PROGRAM Alias
VAR
END_VAR

//R1 & R2 : MCP**  
	//DI
	MCP_IO.MasterStopPB_Pressed					:= NOT Input.R1_01_00;  //NC - Master stop PB not pressed - black pb on mcp
	MCP_IO.CageEstopCircuitOK					:= Input.R1_01_01;  //case Estop circuit okay (Rly1 (120vac)
	MCP_IO.AutoModeSelected						:= Input.R1_01_02; // 0 = manual, 1=auto
	MCP_IO.PSU1_DCOK							:= Input.R1_01_03; //psu1 dc ok
	MCP_IO.MachineGNDrlyOpen					:= Input.R1_01_04; // machine ground lifted (opto board)	
	MCP_IO.CloseAllChargeRlyCommand				:= Input.R1_01_05; // command from screen room (opto)
	MCP_IO.OpenAllDumpRelayCommand				:= Input.R1_01_06; // command from screen room (opto)
	
	MCP_IO.Charger[1].inhibited					:= Input.R1_02_00; //TDK802 1
	MCP_IO.Charger[1].EndOfCharge				:= Input.R1_02_01; //TDK802 1
	MCP_IO.Charger[1].HV_isON					:= Input.R1_02_02; //TDK802 1
	MCP_IO.Charger[1].OverTemp					:= Input.R1_02_03; //TDK802 1
	MCP_IO.Charger[1].InterlockOpen				:= Input.R1_02_04; //TDK802 1
	MCP_IO.Charger[1].LoadFaulted				:= Input.R1_02_05; //TDK802 1
	MCP_IO.Charger[1].SummaryFaulted			:= Input.R1_02_06; //TDK802 1
	
	MCP_IO.Charger[2].inhibited					:= Input.R1_03_00; //TDK802 2
	MCP_IO.Charger[2].EndOfCharge				:= Input.R1_03_01; 
	MCP_IO.Charger[2].HV_isON					:= Input.R1_03_02; 
	MCP_IO.Charger[2].OverTemp					:= Input.R1_03_03; 
	MCP_IO.Charger[2].InterlockOpen				:= Input.R1_03_04; 
	MCP_IO.Charger[2].LoadFaulted				:= Input.R1_03_05; 
	MCP_IO.Charger[2].SummaryFaulted			:= Input.R1_03_06; 
	
	MCP_IO.Charger[3].inhibited					:= Input.R1_04_00; //TDK802 3
	MCP_IO.Charger[3].EndOfCharge				:= Input.R1_04_01; 
	MCP_IO.Charger[3].HV_isON					:= Input.R1_04_02; 
	MCP_IO.Charger[3].OverTemp					:= Input.R1_04_03; 
	MCP_IO.Charger[3].InterlockOpen				:= Input.R1_04_04; 
	MCP_IO.Charger[3].LoadFaulted				:= Input.R1_04_05; 
	MCP_IO.Charger[3].SummaryFaulted			:= Input.R1_04_06; 
	
	MCP_IO.Charger[4].inhibited					:= Input.R1_05_00; //TDK802 4
	MCP_IO.Charger[4].EndOfCharge				:= Input.R1_05_01; 
	MCP_IO.Charger[4].HV_isON					:= Input.R1_05_02; 
	MCP_IO.Charger[4].OverTemp					:= Input.R1_05_03; 
	MCP_IO.Charger[4].InterlockOpen				:= Input.R1_05_04; 
	MCP_IO.Charger[4].LoadFaulted				:= Input.R1_05_05; 
	MCP_IO.Charger[4].SummaryFaulted			:= Input.R1_05_06; 

	MCP_IO.Charger[5].inhibited					:= Input.R1_06_00; //TDK802 5
	MCP_IO.Charger[5].EndOfCharge				:= Input.R1_06_01; 
	MCP_IO.Charger[5].HV_isON					:= Input.R1_06_02; 
	MCP_IO.Charger[5].OverTemp					:= Input.R1_06_03; 
	MCP_IO.Charger[5].InterlockOpen				:= Input.R1_06_04; 
	MCP_IO.Charger[5].LoadFaulted				:= Input.R1_06_05; 
	MCP_IO.Charger[5].SummaryFaulted			:= Input.R1_06_06; 

	MCP_IO.Charger[6].inhibited					:= Input.R1_07_00; //TDK802 6
	MCP_IO.Charger[6].EndOfCharge				:= Input.R1_07_01; 
	MCP_IO.Charger[6].HV_isON					:= Input.R1_07_02; 
	MCP_IO.Charger[6].OverTemp					:= Input.R1_07_03; 
	MCP_IO.Charger[6].InterlockOpen				:= Input.R1_07_04; 
	MCP_IO.Charger[6].LoadFaulted				:= Input.R1_07_05; 
	MCP_IO.Charger[6].SummaryFaulted			:= Input.R1_07_06; 

	MCP_IO.Charger[7].inhibited					:= Input.R1_08_00; //TDK802 7
	MCP_IO.Charger[7].EndOfCharge				:= Input.R1_08_01; 
	MCP_IO.Charger[7].HV_isON					:= Input.R1_08_02; 
	MCP_IO.Charger[7].OverTemp					:= Input.R1_08_03; 
	MCP_IO.Charger[7].InterlockOpen				:= Input.R1_08_04; 
	MCP_IO.Charger[7].LoadFaulted				:= Input.R1_08_05; 
	MCP_IO.Charger[7].SummaryFaulted			:= Input.R1_08_06; 

	MCP_IO.Charger[8].inhibited					:= Input.R1_09_00; //TDK802 8
	MCP_IO.Charger[8].EndOfCharge				:= Input.R1_09_01; 
	MCP_IO.Charger[8].HV_isON					:= Input.R1_09_02; 
	MCP_IO.Charger[8].OverTemp					:= Input.R1_09_03; 
	MCP_IO.Charger[8].InterlockOpen				:= Input.R1_09_04; 
	MCP_IO.Charger[8].LoadFaulted				:= Input.R1_09_05; 
	MCP_IO.Charger[8].SummaryFaulted			:= Input.R1_09_06; 

	//AI
	MCP_IO.Charger[1].voltageFeedback_raw		:= Input.R2_03_00;
	MCP_IO.Charger[1].currentFeedback_raw		:= Input.R2_03_01;
	MCP_IO.Charger[2].voltageFeedback_raw		:= Input.R2_03_02;
	MCP_IO.Charger[2].currentFeedback_raw		:= Input.R2_03_03;
	MCP_IO.Charger[3].voltageFeedback_raw		:= Input.R2_03_04;
	MCP_IO.Charger[3].currentFeedback_raw		:= Input.R2_03_05;
	MCP_IO.Charger[4].voltageFeedback_raw		:= Input.R2_03_06;
	MCP_IO.Charger[4].currentFeedback_raw		:= Input.R2_03_07;
	MCP_IO.Charger[5].voltageFeedback_raw		:= Input.R2_04_00;
	MCP_IO.Charger[5].currentFeedback_raw		:= Input.R2_04_01;
	MCP_IO.Charger[6].voltageFeedback_raw		:= Input.R2_04_02;
	MCP_IO.Charger[6].currentFeedback_raw		:= Input.R2_04_03;
	MCP_IO.Charger[7].voltageFeedback_raw		:= Input.R2_04_04;
	MCP_IO.Charger[7].currentFeedback_raw		:= Input.R2_04_05;
	MCP_IO.Charger[8].voltageFeedback_raw		:= Input.R2_04_06;
	MCP_IO.Charger[8].currentFeedback_raw		:= Input.R2_04_07;
	
	//DQ
	Output.R2_01_00	:= MCP_IO.Charger[1].inhibit;
	Output.R2_01_01	:= MCP_IO.Charger[1].HV_ON;
	Output.R2_01_02	:= MCP_IO.Charger[2].inhibit;
	Output.R2_01_03	:= MCP_IO.Charger[2].HV_ON;
	Output.R2_01_04	:= MCP_IO.Charger[3].inhibit;
	Output.R2_01_05	:= MCP_IO.Charger[3].HV_ON;
	Output.R2_01_06	:= MCP_IO.Charger[4].inhibit;
	Output.R2_01_07	:= MCP_IO.Charger[4].HV_ON;
	
	Output.R2_02_00	:= MCP_IO.Charger[5].inhibit;
	Output.R2_02_01	:= MCP_IO.Charger[5].HV_ON;
	Output.R2_02_02	:= MCP_IO.Charger[6].inhibit;
	Output.R2_02_03	:= MCP_IO.Charger[6].HV_ON;
	Output.R2_02_04	:= MCP_IO.Charger[7].inhibit;
	Output.R2_02_05	:= MCP_IO.Charger[7].HV_ON;
	Output.R2_02_06	:= MCP_IO.Charger[8].inhibit;
	Output.R2_02_07	:= MCP_IO.Charger[8].HV_ON;
	
	Output.R2_06_00	:= MCP_IO.GLS1_hvON;
	Output.R2_06_01	:= MCP_IO.GLS2_hvON;
	Output.R2_06_02	:= MCP_IO.GLS3_hvON;
	Output.R2_06_03	:= MCP_IO.LiftMachineGND;
	Output.R2_06_04	:= MCP_IO.AllChargeRelaysClose; //only for slim
	Output.R2_06_05	:= MCP_IO.AllDumpRelaysOpen;  // only for slim
	
	//AQ
	Output.R2_05_00	:= MCP_IO.Charger[1].voltageSP;
	Output.R2_05_01	:= MCP_IO.Charger[2].voltageSP;
	Output.R2_05_02	:= MCP_IO.Charger[3].voltageSP;
	Output.R2_05_03	:= MCP_IO.Charger[4].voltageSP;	
	Output.R2_05_04	:= MCP_IO.Charger[5].voltageSP;
	Output.R2_05_05	:= MCP_IO.Charger[6].voltageSP;
	Output.R2_05_06	:= MCP_IO.Charger[7].voltageSP;
	Output.R2_05_07	:= MCP_IO.Charger[8].voltageSP;					
	
	Output.R2_07_00	:= MCP_IO.GLS1_voltageSP; //Form Trigger
	Output.R2_07_01	:= MCP_IO.GLS2_voltageSP;  //Preform trigger
	Output.R2_07_02	:= MCP_IO.GLS3_voltageSP; //preform cap charger

//R3 : Bank 1 (LCP1)***********************************************
	//EL3068 - AI
	LCP.Section[1].Peak.cap[1].voltageFeedback_raw := Input.R3_01_00;
	LCP.Section[1].Peak.cap[2].voltageFeedback_raw := Input.R3_01_01;
	LCP.Section[1].Peak.cap[3].voltageFeedback_raw := Input.R3_01_02;
	LCP.Section[1].Peak.cap[4].voltageFeedback_raw := Input.R3_01_03;
	LCP.Section[1].Peak.cap[5].voltageFeedback_raw := Input.R3_01_04;
	LCP.Section[1].Peak.cap[6].voltageFeedback_raw := Input.R3_01_05;
	LCP.Section[1].Peak.cap[7].voltageFeedback_raw := Input.R3_01_06;
	LCP.Section[1].Peak.cap[8].voltageFeedback_raw := Input.R3_01_07;
	LCP.Section[1].Peak.cap[9].voltageFeedback_raw := Input.R3_02_00;
	LCP.Section[1].Peak.cap[10].voltageFeedback_raw := Input.R3_02_01;
	
	LCP.Section[1].Sust.cap[1].voltageFeedback_raw := Input.R3_02_02;
	LCP.Section[1].Sust.cap[2].voltageFeedback_raw := Input.R3_02_03;
	
	//DI
	LCP.Section[1].Peak.ChargeRelay1_close 	:= Input.R3_03_00; //RLY 1A
	LCP.Section[1].Peak.ChargeRelay2_close 	:= Input.R3_03_01; //RLY 2A
	LCP.Section[1].Peak.DumpRelay1_close 	:= Input.R3_03_02; //RLY 3A
	LCP.Section[1].Peak.DumpRelay2_close	:= Input.R3_03_03; //RLY 4A
	LCP.Section[1].Sust.ChargeRelay1_close	:= Input.R3_03_04; //RLY 5A
	LCP.Section[1].Sust.ChargeRelay2_close	:= Input.R3_03_05; //RLY 6A
	LCP.Section[1].Sust.DumpRelay1_close	:= Input.R3_03_06; //RLY 7A
	LCP.Section[1].Sust.DumpRelay2_close	:= Input.R3_03_07; //RLY 8A
	
	LCP.Section[1].Peak.ShortContact1_close 	:= Input.R3_04_00; //psw1
	LCP.Section[1].Peak.UnshortContact1_close 	:= Input.R3_04_01; //psw2
	LCP.Section[1].Peak.ShortContact2_close 	:= Input.R3_04_02; //psw3
	LCP.Section[1].Peak.UnshortContact2_close 	:= Input.R3_04_03; //psw4
	LCP.Section[1].LossPneumaticPressure 		:= Input.R3_04_04; //psw5
	LCP.Section[1].PSU1_DCOK					:= Input.R3_04_05; //psu1 contact

	//DQ
	Output.R3_05_00 := LCP.Section[1].Peak.CloseChargeRelay1; //RLY1
	Output.R3_05_01 := LCP.Section[1].Peak.CloseChargeRelay2; //RLY2
	Output.R3_05_02 := LCP.Section[1].Peak.OpenDumpRelay1; //RLY3
	Output.R3_05_03 := LCP.Section[1].Peak.OpenDumpRelay2; //RLY4
	Output.R3_05_04 := LCP.Section[1].Sust.CloseChargeRelay1; //RLY5
	Output.R3_05_05 := LCP.Section[1].Sust.CloseChargeRelay2; //RLY6
	Output.R3_05_06 := LCP.Section[1].Sust.OpenDumpRelay1; //RLY7
	Output.R3_05_07 := LCP.Section[1].Sust.OpenDumpRelay2; //RLY8
	Output.R3_06_00 := LCP.Section[1].SystemReadyToCharge; //LED1

//R4 : Bank 2 (LCP2)***********************************************
	//EL3068 - AI
	LCP.Section[2].Peak.cap[1].voltageFeedback_raw := Input.R4_01_00;
	LCP.Section[2].Peak.cap[2].voltageFeedback_raw := Input.R4_01_01;
	LCP.Section[2].Peak.cap[3].voltageFeedback_raw := Input.R4_01_02;
	LCP.Section[2].Peak.cap[4].voltageFeedback_raw := Input.R4_01_03;
	LCP.Section[2].Peak.cap[5].voltageFeedback_raw := Input.R4_01_04;
	LCP.Section[2].Peak.cap[6].voltageFeedback_raw := Input.R4_01_05;
	LCP.Section[2].Peak.cap[7].voltageFeedback_raw := Input.R4_01_06;
	LCP.Section[2].Peak.cap[8].voltageFeedback_raw := Input.R4_01_07;
	LCP.Section[2].Peak.cap[9].voltageFeedback_raw := Input.R4_02_00;
	LCP.Section[2].Peak.cap[10].voltageFeedback_raw := Input.R4_02_01;
	
	LCP.Section[2].Sust.cap[1].voltageFeedback_raw := Input.R4_02_02;
	LCP.Section[2].Sust.cap[2].voltageFeedback_raw := Input.R4_02_03;
	
	//DI
	LCP.Section[2].Peak.ChargeRelay1_close 	:= Input.R4_03_00; //RLY 1A
	LCP.Section[2].Peak.ChargeRelay2_close 	:= Input.R4_03_01; //RLY 2A
	LCP.Section[2].Peak.DumpRelay1_close 	:= Input.R4_03_02; //RLY 3A
	LCP.Section[2].Peak.DumpRelay2_close	:= Input.R4_03_03; //RLY 4A
	LCP.Section[2].Sust.ChargeRelay1_close	:= Input.R4_03_04; //RLY 5A
	LCP.Section[2].Sust.ChargeRelay2_close	:= Input.R4_03_05; //RLY 6A
	LCP.Section[2].Sust.DumpRelay1_close	:= Input.R4_03_06; //RLY 7A
	LCP.Section[2].Sust.DumpRelay2_close	:= Input.R4_03_07; //RLY 8A
	
	LCP.Section[2].Peak.ShortContact1_close 	:= Input.R4_04_00; //psw1
	LCP.Section[2].Peak.UnshortContact1_close 	:= Input.R4_04_01; //psw2
	LCP.Section[2].Peak.ShortContact2_close 	:= Input.R4_04_02; //psw3
	LCP.Section[2].Peak.UnshortContact2_close 	:= Input.R4_04_03; //psw4
	LCP.Section[2].LossPneumaticPressure 		:= Input.R4_04_04; //psw5
	LCP.Section[2].PSU1_DCOK					:= Input.R4_04_05; //psu1 contact

	//DQ
	Output.R4_05_00 := LCP.Section[2].Peak.CloseChargeRelay1; //RLY1
	Output.R4_05_01 := LCP.Section[2].Peak.CloseChargeRelay2; //RLY2
	Output.R4_05_02 := LCP.Section[2].Peak.OpenDumpRelay1; //RLY3
	Output.R4_05_03 := LCP.Section[2].Peak.OpenDumpRelay2; //RLY4
	Output.R4_05_04 := LCP.Section[2].Sust.CloseChargeRelay1; //RLY5
	Output.R4_05_05 := LCP.Section[2].Sust.CloseChargeRelay2; //RLY6
	Output.R4_05_06 := LCP.Section[2].Sust.OpenDumpRelay1; //RLY7
	Output.R4_05_07 := LCP.Section[2].Sust.OpenDumpRelay2; //RLY8
	Output.R4_06_00 := LCP.Section[2].SystemReadyToCharge; //LED1

//R5 : Bank 3 (LCP3)***********************************************
	//EL3068 - AI
	LCP.Section[3].Peak.cap[1].voltageFeedback_raw := Input.R5_01_00;
	LCP.Section[3].Peak.cap[2].voltageFeedback_raw := Input.R5_01_01;
	LCP.Section[3].Peak.cap[3].voltageFeedback_raw := Input.R5_01_02;
	LCP.Section[3].Peak.cap[4].voltageFeedback_raw := Input.R5_01_03;
	LCP.Section[3].Peak.cap[5].voltageFeedback_raw := Input.R5_01_04;
	LCP.Section[3].Peak.cap[6].voltageFeedback_raw := Input.R5_01_05;
	LCP.Section[3].Peak.cap[7].voltageFeedback_raw := Input.R5_01_06;
	LCP.Section[3].Peak.cap[8].voltageFeedback_raw := Input.R5_01_07;
	LCP.Section[3].Peak.cap[9].voltageFeedback_raw := Input.R5_02_00;
	LCP.Section[3].Peak.cap[10].voltageFeedback_raw := Input.R5_02_01;
	
	LCP.Section[3].Sust.cap[1].voltageFeedback_raw := Input.R5_02_02;
	LCP.Section[3].Sust.cap[2].voltageFeedback_raw := Input.R5_02_03;
	
	//DI
	LCP.Section[3].Peak.ChargeRelay1_close 	:= Input.R5_03_00; //RLY 1A
	LCP.Section[3].Peak.ChargeRelay2_close 	:= Input.R5_03_01; //RLY 2A
	LCP.Section[3].Peak.DumpRelay1_close 	:= Input.R5_03_02; //RLY 3A
	LCP.Section[3].Peak.DumpRelay2_close	:= Input.R5_03_03; //RLY 4A
	LCP.Section[3].Sust.ChargeRelay1_close	:= Input.R5_03_04; //RLY 5A
	LCP.Section[3].Sust.ChargeRelay2_close	:= Input.R5_03_05; //RLY 6A
	LCP.Section[3].Sust.DumpRelay1_close	:= Input.R5_03_06; //RLY 7A
	LCP.Section[3].Sust.DumpRelay2_close	:= Input.R5_03_07; //RLY 8A
	
	LCP.Section[3].Peak.ShortContact1_close 	:= Input.R5_04_00; //psw1
	LCP.Section[3].Peak.UnshortContact1_close 	:= Input.R5_04_01; //psw2
	LCP.Section[3].Peak.ShortContact2_close 	:= Input.R5_04_02; //psw3
	LCP.Section[3].Peak.UnshortContact2_close 	:= Input.R5_04_03; //psw4
	LCP.Section[3].LossPneumaticPressure 		:= Input.R5_04_04; //psw5
	LCP.Section[3].PSU1_DCOK					:= Input.R5_04_05; //psu1 contact

	//DQ
	Output.R5_05_00 := LCP.Section[3].Peak.CloseChargeRelay1; //RLY1
	Output.R5_05_01 := LCP.Section[3].Peak.CloseChargeRelay2; //RLY2
	Output.R5_05_02 := LCP.Section[3].Peak.OpenDumpRelay1; //RLY3
	Output.R5_05_03 := LCP.Section[3].Peak.OpenDumpRelay2; //RLY4
	Output.R5_05_04 := LCP.Section[3].Sust.CloseChargeRelay1; //RLY5
	Output.R5_05_05 := LCP.Section[3].Sust.CloseChargeRelay2; //RLY6
	Output.R5_05_06 := LCP.Section[3].Sust.OpenDumpRelay1; //RLY7
	Output.R5_05_07 := LCP.Section[3].Sust.OpenDumpRelay2; //RLY8
	Output.R5_06_00 := LCP.Section[3].SystemReadyToCharge; //LED1

//R6 : Bank 4 (LCP4)*****Formation******************************************
	//EL3068 - AI
	LCP.Section[4].Form.cap[1].voltageFeedback_raw := Input.R6_01_00;
	LCP.Section[4].Form.cap[2].voltageFeedback_raw := Input.R6_01_01;
	LCP.Section[4].Form.cap[3].voltageFeedback_raw := Input.R6_01_02;
	LCP.Section[4].Form.cap[4].voltageFeedback_raw := Input.R6_01_03;
	LCP.Section[4].Form.cap[5].voltageFeedback_raw := Input.R6_01_04;
	LCP.Section[4].Form.cap[6].voltageFeedback_raw := Input.R6_01_05;
	LCP.Section[4].Form.cap[7].voltageFeedback_raw := Input.R6_01_06;
	LCP.Section[4].Form.cap[8].voltageFeedback_raw := Input.R6_01_07;
	
	LCP.Section[4].Form.cap[9].voltageFeedback_raw	:= Input.R6_02_00;
	LCP.Section[4].Form.cap[10].voltageFeedback_raw := Input.R6_02_01;
	LCP.Section[4].Form.cap[11].voltageFeedback_raw := Input.R6_02_02;
	LCP.Section[4].Form.cap[12].voltageFeedback_raw := Input.R6_02_03;
	LCP.Section[4].FormTriggerCapVoltage_raw		 := Input.R6_02_04;
	
	//DI
	LCP.Section[4].Form.ChargeRelay1_close			:= Input.R6_03_00;	//RLY 1A
	LCP.Section[4].Form.ChargeRelay2_close			:= Input.R6_03_01;	//RLY 2A
	LCP.Section[4].Form.PreFormChargeRly_close		:= Input.R6_03_02;	//RLY 3A	
	LCP.Section[4].Form.FormTrigChargeRly_close		:= Input.R6_03_03;	//RLY 4A
	LCP.Section[4].Form.PreFormTrigChargeRly_close	:= Input.R6_03_04;	//RLY 5A
	LCP.Section[4].Form.DumpRelay1_close			:= Input.R6_03_05;	//RLY 6A
	LCP.Section[4].Form.DumpRelay2_close			:= Input.R6_03_06;	//RLY 7A
	LCP.Section[4].Form.PreFormDumpRly_close		:= Input.R6_03_07;	//RLY 8A
	LCP.Section[4].Form.FormTrigDumpRly1_close		:= Input.R6_04_00;	//RLY 9A
	LCP.Section[4].Form.PreFormTrigDumpRly1_close	:= Input.R6_04_01;	//RLY 10A
	
	LCP.Section[4].Form.ShortContact1_close		:= Input.R6_04_02;  //psw1
	LCP.Section[4].Form.UnshortContact1_close	:= Input.R6_04_03;  //psw2
	LCP.Section[4].Form.ShortContact2_close		:= Input.R6_04_04;  //psw3
	LCP.Section[4].Form.UnshortContact2_close	:= Input.R6_04_05;  //psw4
	LCP.Section[4].Form.FormTrigShortContact_close		:= Input.R6_04_06;  //psw5
	LCP.Section[4].Form.FormTrigUnshortContact_close	:= Input.R6_04_07;  //psw6
	LCP.Section[4].Form.PreFormTrigShortContact_close	:= Input.R6_05_00;  //psw7
	LCP.Section[4].Form.PreFormTrigUnShortContact_close	:= Input.R6_05_01;  //psw8
	LCP.Section[4].LossPneumaticPressure				:= Input.R6_05_02;  //psw9
	LCP.Section[4].PSU1_DCOK							:= Input.R6_05_03;  //psu1
	
	//DQ
	Output.R6_06_00 := LCP.Section[4].Form.CloseChargeRelay1; //rly1
	Output.R6_06_01 := LCP.Section[4].Form.CloseChargeRelay2; //rly2
	Output.R6_06_02 := LCP.Section[4].Form.ClosePreFormChargeRly; //rly3
	Output.R6_06_03 := LCP.Section[4].Form.CloseFormTrigChargeRly; //rly4
	Output.R6_06_04 := LCP.Section[4].Form.ClosePreFormTrigChargeRly; //rly5
	Output.R6_06_05 := LCP.Section[4].Form.OpenDumpRelay1; //rly6
	Output.R6_06_06 := LCP.Section[4].Form.OpenDumpRelay2; //rly7
	Output.R6_06_07 := LCP.Section[4].Form.OpenPreFormDumpRly; //rly8
	
	Output.R6_07_00 := LCP.Section[4].Form.OpenFormTrigDumpRly1; //rly9
	Output.R6_07_01 := LCP.Section[4].Form.OpenPreFormTrigDumpRly1; //rly10
	Output.R6_07_02 := LCP.Section[4].SystemReadyToCharge; //LED1
	
	//InstrumentReading.R2_01_CH00 := Input.R3_01_00;
	//InstrumentReading.R2_01_CH01 := Input.R3_01_01;
	(*
	R2_01_02 		AT %I*: INT;
	R2_01_02_Status AT %I*: WORD;
	
	R2_01_03 		AT %I*: INT;
	R2_01_03_Status AT %I*: WORD;
	
	R2_01_04 		AT %I*: INT;
	R2_01_04_Status AT %I*: WORD;
	
	R2_01_05 		AT %I*: INT;
	R2_01_05_Status AT %I*: WORD;
	
	R2_01_06 		AT %I*: INT;
	R2_01_06_Status AT %I*: WORD;
	
	R2_01_07 		AT %I*: INT;
	R2_01_07_Status AT %I*: WORD;
	*)

END_PROGRAM

(* stored: Version 1.1.0.1, ProductVersion 3.1.4024.11
   POU Alias: Id {ebc75665-f0df-4b03-b4d1-48515468f179}, SpecialFunc None *)
